// TwinCAT 3 PLC project Python_SPS
// ProgramVersion: 3.1.4024.0
// libraries:
//   Tc2_Standard, * (Beckhoff Automation GmbH)
//   Tc2_System, * (Beckhoff Automation GmbH)
//   Tc3_Module, * (Beckhoff Automation GmbH)
// project tree:
//   / PlcTask.TcTTO
//   POUs/ MAIN.TcPOU
//   Python/ MAIN_LIB_Python.TcPOU
//   Python/Privat/DUTs/ Python_Kamera_Daten_Kommando.TcDUT, Python_Kamera_Daten_Status.TcDUT, Python_Kamera_Interface.TcDUT
//   Python/Public/Config/ Python_Kamera_Liste.TcDUT
//   Python/Public/DUTs/ Python_Checker.TcDUT, Python_Kamera_Daten.TcDUT, Parameter.TcDUT, Parameter_Lokal.TcDUT
//   Python/Public/GVLs/ GVL_Python_Kamera.TcGVL
//   Python/Public/POUs/ POU_Auto_Trigger_Kamera.TcPOU, Python_Checker_Modul.TcPOU
// real-time tasks:
//   TASK PlcTask: cycle T#10ms, priority 20, ADS port 350

CONFIGURATION Python_SPS
    RESOURCE PLC ON TwinCAT3
        TASK PlcTask(INTERVAL := T#10ms, PRIORITY := 20);
        PROGRAM MAIN WITH PlcTask : MAIN;
    END_RESOURCE
END_CONFIGURATION

// ---- Python/Privat/DUTs/Python_Kamera_Daten_Kommando.TcDUT
TYPE Python_Kamera_Daten_Kommando :
STRUCT
		
		Trigger				:BOOL;
		ID					:STRING(32);
		Wafer_Type			:INT; 			
		
END_STRUCT
END_TYPE

// ---- Python/Privat/DUTs/Python_Kamera_Daten_Status.TcDUT
TYPE Python_Kamera_Daten_Status :
STRUCT
	
	 Busy						:BOOL;
	 IsDone						:BOOL;
	 PictureValid				:BOOL;
	 Active						:BOOL; 
 
END_STRUCT
END_TYPE

// ---- Python/Privat/DUTs/Python_Kamera_Interface.TcDUT
TYPE Python_Kamera_Interface :
	STRUCT
		
		CameraName		:STRING(32);
		CMD				: Python_Kamera_Daten_Kommando;
		STAT			: Python_Kamera_Daten_Status;
		
	END_STRUCT
END_TYPE

// ---- Python/Public/Config/Python_Kamera_Liste.TcDUT

TYPE Python_Kamera_Liste :
(
	Python_Kamera_Liste_Untergrenze,
	Python_Kamera_Liste_01,
	Python_Kamera_Liste_02,
	Python_Kamera_Liste_03,
	Python_Kamera_Liste_Obergrenze
);
END_TYPE

// ---- Python/Public/DUTs/Python_Checker.TcDUT
TYPE Python_Checker :
STRUCT
		
		Python_Active			:BOOL := FALSE;
		Test					:BOOL := FALSE;
		Python_ERROR			:BOOL := FALSE;

END_STRUCT
END_TYPE

// ---- Python/Public/DUTs/Python_Kamera_Daten.TcDUT
TYPE Python_Kamera_Daten :
STRUCT
	
	Lokal		: ARRAY [Python_Kamera_Liste_Untergrenze..Python_Kamera_Liste_Obergrenze] OF  Python_Kamera_Interface;
	
END_STRUCT
END_TYPE

// ---- Python/Public/DUTs/Parameter.TcDUT
TYPE Parameter :
STRUCT
	
	Lokal		: ARRAY [Python_Kamera_Liste_Untergrenze..Python_Kamera_Liste_Obergrenze] OF  Parameter_Lokal;
	
END_STRUCT
END_TYPE

// ---- Python/Public/DUTs/Parameter_Lokal.TcDUT
TYPE Parameter_Lokal :
STRUCT
	
	Name				:STRING(32);
	Value				:TIME;
	
END_STRUCT
END_TYPE

// ---- Python/Public/GVLs/GVL_Python_Kamera.TcGVL
{attribute 'Tc2GvlVarNames'}
VAR_GLOBAL
	
	Python_Kamera_Anzahl	: INT := Python_Kamera_Liste_Obergrenze - 1; 
	Python_Checker			: Python_Checker;
	
	//Kameradaten werden initalisiert und die Namen für die Kameras festgelegt	
	Python_Kamera_Daten 	: Python_Kamera_Daten
		
		:= (
				Lokal:=
					[
						(* Unbelegt MUSS als erster Eintrag vorhanden sein *)
						(),
						(* Kamera_CAM1 *)
						( CameraName := 'Kamera_CAM1'),
						(* Kamera_CAM2 *)
						( CameraName := 'Kamera_CAM2'),
						(* Kamera_CAM3 *)
						( CameraName := 'Kamera_CAM3'),
						(* Obergrenze *)
						()
					]
				);
				
	// Hier werden die Parameter festgelegt
	Parameter		: Parameter
		
		:= (
				Lokal:=
					[
						(* Unbelegt MUSS als erster Eintrag vorhanden sein *)
						(),
						(* Kamera_CAM1 *)
						( Name:= 'Kamera_CAM1', Value := T#4S),
						(* Kamera_CAM2 *)
						( Name:= 'Kamera_CAM2', Value := T#2S),
						(* Kamera_CAM3 *)
						( Name:= 'Kamera_CAM3', Value := T#8S),
						(* Obergrenze *)
						()
					]
				);
				
		
		
			
END_VAR

// ---- POUs/MAIN.TcPOU
PROGRAM MAIN
VAR
END_VAR

MAIN_LIB_Python();

END_PROGRAM

// ---- Python/MAIN_LIB_Python.TcPOU
PROGRAM MAIN_LIB_Python
VAR
	L_Kamera_Index						: INT;
	L_Python_Checker					: Python_Checker_Modul;
	L_POU_Auto_Trigger_Kamera			: ARRAY [Python_Kamera_Liste_Untergrenze..Python_Kamera_Liste_Obergrenze] OF POU_Auto_Trigger_Kamera;
END_VAR


L_Python_Checker(
	EA_Python_Checker		:= Python_Checker
);


FOR L_Kamera_Index := Python_Kamera_Liste_Untergrenze + 1  TO Python_Kamera_Liste_Obergrenze - 1 DO	(* $JR_Kamera_VisionX1.3.0$ *)

	L_POU_Auto_Trigger_Kamera[L_Kamera_Index](
		
		EA_Kamera_Index		:= L_Kamera_Index
		
	);

END_FOR

END_PROGRAM

// ---- Python/Public/POUs/Python_Checker_Modul.TcPOU
FUNCTION_BLOCK Python_Checker_Modul
VAR_IN_OUT
	
		EA_Python_Checker			: Python_Checker;
END_VAR
VAR
		
		TON_1						:TON;
		TON_2						:TON;
END_VAR



IF EA_Python_Checker.Python_Active THEN
	TON_1(IN := TRUE, PT := T#5000MS);

	IF TON_1.Q THEN
		EA_Python_Checker.Test := TRUE;
		TON_1(In := FALSE);
	END_IF

	TON_2(IN := EA_Python_Checker.Test, PT := T#5000MS);

	IF TON_2.Q THEN 
		EA_Python_Checker.Python_ERROR := TRUE;
		EA_Python_Checker.Python_Active := FALSE;
		TON_2(In := FALSE);
	END_IF
	
ELSE
	TON_1(In := FALSE);
	EA_Python_Checker.Test := FALSE; 


END_IF

END_FUNCTION_BLOCK

// ---- Python/Public/POUs/POU_Auto_Trigger_Kamera.TcPOU
FUNCTION_BLOCK POU_Auto_Trigger_Kamera

VAR_INPUT
	
		EA_Kamera_Index			: INT;
END_VAR

VAR
	
	//Locale Variablen
	L_Enable: 					BOOL;
	L_TEMP_CAM_ID: 				INT;
	L_Step_ID: 					INT := 0;
	L_SUCCESS:					BOOL;
	L_Done:						BOOL;
	L_Test_ID: 					INT := 1;
	L_Delay_TON : 				TON;
	L_Error_TON : 				TON;
	
END_VAR

IF NOT L_Enable THEN
	L_Step_ID := 0;
	RETURN;
END_IF

CASE L_Step_ID OF
	
0:
	//1. Überprüfen ob Kamera bereit ist, falls ja Trigger senden
	L_Error_TON(IN := TRUE, PT:= T#5S);
	
	L_SUCCESS := Python_Kamera_Daten.Lokal[EA_Kamera_Index].STAT.Active AND
					Python_Checker.Python_Active AND
					NOT Python_Kamera_Daten.Lokal[EA_Kamera_Index].STAT.Busy; 
	IF L_SUCCESS THEN
		Python_Kamera_Daten.Lokal[EA_Kamera_Index].CMD.ID := CONCAT('Test_', INT_TO_STRING(L_Test_ID));
		Python_Kamera_Daten.Lokal[EA_Kamera_Index].CMD.Trigger := TRUE;
		
		// Hier wird STAT von Regime
		Python_Kamera_Daten.Lokal[EA_Kamera_Index].STAT.IsDone := FALSE;
		Python_Kamera_Daten.Lokal[EA_Kamera_Index].STAT.PictureValid := FALSE;
		//
		
		L_Error_TON(IN:=FALSE);
		L_Step_ID := 10;
	END_IF
	
	IF L_Error_TON.Q THEN
		L_Error_TON(IN:=FALSE);
		L_Step_ID := 100;	
	END_IF
	
10:
	//2. Überprüfe ob das Bild valide war und ob der Auftrag abgeschlossen ist
	L_Error_TON(IN := TRUE, PT:= T#5S);
	
	L_Done :=  Python_Kamera_Daten.Lokal[EA_Kamera_Index].STAT.IsDone AND
					Python_Kamera_Daten.Lokal[EA_Kamera_Index].STAT.PictureValid AND
					NOT Python_Kamera_Daten.Lokal[EA_Kamera_Index].STAT.Busy ;
	IF L_DONE THEN
		L_Step_ID := 20;
		L_Error_TON(IN:=FALSE);
	END_IF
	
	IF L_Error_TON.Q THEN
		L_Error_TON(IN:=FALSE);
		L_Step_ID := 100;	
	END_IF

20:
	//3. Trigger zurücksetzen
	Python_Kamera_Daten.Lokal[EA_Kamera_Index].CMD.Trigger := FALSE;
	//Increase Test ID
	L_Test_ID := L_Test_ID + 1;
	IF L_Test_ID > 100 THEN
		L_Test_ID := 1;
	END_IF
	L_Step_ID := 30;
	
30:
 	//4. ein kleiner delay,sodass nur alle 2 sekunden getriggert wird
 	L_Delay_TON(IN := TRUE, PT := Parameter.Lokal[EA_Kamera_Index].Value);
	
	IF L_Delay_TON.Q THEN
		L_Delay_TON(IN:= FALSE);
		L_Step_ID := 0;
	END_IF
	
100:
	L_Enable := FALSE;
	Python_Checker.Python_ERROR := TRUE;
	
	
	
	

END_CASE

END_FUNCTION_BLOCK
